TYPE ST_MachinePreparationConfig :
STRUCT
    //==========================================================
    // 整机准备位置
    //==========================================================
    fTrayXStandby       : LREAL;
    fTrayZStandby       : LREAL;

    fDamperXStandby     : LREAL;
    fDamperYStandby     : LREAL;
    fDamperZStandby     : LREAL;
    fDamperRotationZero : LREAL;

    fClampOpenPosition  : LREAL;
    fTurntableZero      : LREAL;
	// 同轴度调整机构准备位置
	fAdjustmentXStandby : LREAL;
	fAdjustmentYStandby : LREAL;
	fAdjustmentZStandby : LREAL;
	
    fScrewdriverYZero   : LREAL;
    fScrewdriverZSafe   : LREAL;

    //==========================================================
    // 速度
    //==========================================================
    fTrayVelocity           : LREAL;
    fDamperVelocity         : LREAL;
    fDamperRotationVelocity : LREAL;
    fClampVelocity          : LREAL;
    fTurntableVelocity      : LREAL;
	fAdjustmentVelocity 	: LREAL;
    fScrewdriverVelocity    : LREAL;

    //==========================================================
    // 到位公差与超时
    //==========================================================
    fLinearTolerance   : LREAL;
    fRotationTolerance : LREAL;

    tReadyTimeout      : TIME;
    tMotionTimeout     : TIME;
    // 仅传输既有配置源，不设置第二套默认数值。
    fTrayRackStationX : LREAL;
    aTrayLayer : ARRAY[1..5] OF ST_TrayLayerPositionConfig;
    fTrayRecoveryBoundaryTolerance : LREAL;
    tTrayRecoveryTimeout : TIME;
    tTrayReleaseConfirmTimeout : TIME;
    tTrayDetectStable : TIME;
END_STRUCT
END_TYPE

(* stored: Version 1.1.0.1, ProductVersion 3.1.4026.20
   DUT ST_MachinePreparationConfig: Id {5a7a8a07-dcd0-48bc-ae3c-f9a00a4914a8} *)
